{attribute 'linkalways'} 
{attribute 'no_explicit_call' := 'This FB is a CLASS and must be accessed using methods or properties'}
{attribute 'enable_dynamic_creation'}
FUNCTION_BLOCK Node_F_VN_FillContainer_TcVnPoint3_REAL EXTENDS VisionNode
VAR
    ipContainer : _ITcVnContainer;
    aValue : _TcVnPoint3_REAL;
    hrPrev : _HRESULT(S_OK);
    hresult : _HRESULT(S_OK);
END_VAR

METHOD PUBLIC  Clone : I_Node
VAR
    pNode : POINTER TO Node_F_VN_FillContainer_TcVnPoint3_REAL;
END_VAR
pNode := __NEW(Node_F_VN_FillContainer_TcVnPoint3_REAL);
Clone := pNode^;
END_METHOD

METHOD FB_init : BOOL
VAR_INPUT
    bInitRetains : BOOL; // if TRUE, the retain variables are initialized (warm start / cold start)
    bInCopyCode : BOOL;  // if TRUE, the instance afterwards gets moved into the copy code (online change)
END_VAR
AddInput('ipContainer', ipContainer);
AddInput('aValue', aValue);
AddInput('hrPrev', hrPrev);
AddOutput('ipContainer', ipContainer);
AddOutput('hresult',hresult);
END_METHOD

METHOD PROTECTED OnExecute : HRESULT
hresult.Value := F_VN_FillContainer_TcVnPoint3_REAL(
    ipContainer := ipContainer.Value,
    aValue := aValue.Value,
    hrPrev:= hrPrev.Value);
END_METHOD

METHOD PUBLIC PreExecutionCheck
VAR_INPUT
    Check : I_PreExecutionChecks;
END_VAR
Check.IsTrue(ipContainer.IsValid, 'ipContainer must be a valid container');
END_METHOD

END_FUNCTION_BLOCK

(* stored: Version 1.1.0.1, ProductVersion 3.1.4024.13
   POU Node_F_VN_FillContainer_TcVnPoint3_REAL: Id {2d0a7f7f-68eb-4f88-a56d-34413a79ec2a}, SpecialFunc None
   Folder Constructor: Id {a88fbe1b-3ee2-458c-98b9-74601d8c0df0}
   Method Clone: Id {ffa46962-5eb6-4b8d-bb2f-3a4eebe1f02d}
   Method FB_init: Id {ff5ab8c3-c54b-4549-8a12-e5266fcb7082}
   Method OnExecute: Id {97419ca5-7eef-4e87-87c3-f0b79f3d2391}
   Method PreExecutionCheck: Id {bf4143e1-9c66-43b6-a110-1bbbc804b769} *)
